// TIA Portal V19 export
FUNCTION "V0101 Condensate Alarms" : Void   // FC102, STL
{ S7_Optimized_Access := 'TRUE' }
// stored: AutoNumber false
   VAR_TEMP
      tmp : Bool;
   END_VAR
BEGIN

NETWORK
TITLE = TT0178 Condensate temperature High
      A(;
      O(;
      L     "MeasuredValues".TT0178REAL;
      L     "SetpointsV0101Condensate".TT0178_CondenseHigh;
      >R;
      );
      O(;
      L     "MeasuredValues".TT0178REAL;
      L     "SetpointsV0101Condensate".TT0178_CondenseLow;
      <R;
      );
      );
      A(;
      A     "IF_Device".V_09_31.IO.V._IO.IN.Activate;
      L     S5T#1M;
      SD    "Tag_101";
      NOP   0;
      NOP   0;
      NOP   0;
      A     "Tag_101";
      );
      S     "ProcessAndPbAlarms"."A"[64];  //A64_TT0178_TempFault

NETWORK
TITLE = TT0930 temperature Low
      A(;
      L     "IF_Device".TTX_09_30.ProcessData.Temperature;
      L     "SetpointsV0101Condensate".TT0930_Low_Prod;
      <R;
      );
      A(;
      A     "Y0906";
      L     S5T#1M;
      SD    "Tag_102";
      NOP   0;
      NOP   0;
      NOP   0;
      A     "Tag_102";
      );
      S     "ProcessAndPbAlarms"."A"[65];  //A65_TT0930_Low

NETWORK
TITLE = TT0931 temperature Low
      A(;
      L     "IF_Device".TTX_09_31.ProcessData.Temperature;
      L     "SetpointsV0101Condensate".TT0931_Low_Prod;
      <R;
      );
      A(;
      A     "Y0148";
      AN    "Y0103";
      AN    "Y0104";
      L     S5T#1M;
      SD    "Tag_103";
      NOP   0;
      NOP   0;
      NOP   0;
      A     "Tag_103";
      );
      S     "ProcessAndPbAlarms"."A"[67];  //A67_TT0931_Low

NETWORK
TITLE = V0101 Changing
      A(;
      A(;
      A     "Y0101";
      FP    "Tag_104";
      O(;
      A     "Y0101";
      FN    "Tag_105";
      );
      );
      S     "M15.0";
      A     "Tag_106";
      R     "M15.0";
      A     "M15.0";
      );
      L     S5T#1M;
      SD    "Tag_106";
      NOP   0;
      NOP   0;
      NOP   0;
      A     "Tag_106";
      =     #tmp;

NETWORK
TITLE = CT0930 Condensate Conductivity High
      A(;
      L     "IF_Device".CTX_09_30.ProcessData.Conductivity;
      L     "SetpointsV0101Condensate".CT0930_High;
      >R;
      );
      A(;
      A     "IF_Device".V_09_31.IO.V._IO.IN.Activate;
      AN    "M15.0";
      L     S5T#1M;
      SD    "Tag_107";
      NOP   0;
      NOP   0;
      NOP   0;
      A     "Tag_107";
      );
      S     "ProcessAndPbAlarms"."A"[68];  //A68_CT0930_High
END_FUNCTION
